// TIA Portal V17 export
// export: Created 2025-05-06T13:48:25.8957092Z, ExportSetting WithDefaults, DisplayName Totally Integrated Automation Portal, DisplayVersion V17 Update 8, DisplayName TIA Portal Openness, DisplayVersion V17 Update 8, DisplayName TIA Portal Version Control Interface, DisplayVersion V17, DisplayName SINAMICS Startdrive Advanced, DisplayVersion V17 SP2, DisplayName SINAMICS Startdrive G110M, G120, G120C, G120D, G120P, G115D, DisplayVersion V17 SP2, DisplayName SINAMICS Startdrive G130, G150, S120, S150, SINAMICS MV, S210, DisplayVersion V17 SP2, DisplayName STEP 7 Professional, DisplayVersion V17 Update 8, DisplayName SINUMERIK ONE STEP 7 Toolbox, DisplayVersion V17 Update 12, DisplayName SINUMERIK 840D sl STEP 7 Toolbox, DisplayVersion V17 Update 12, DisplayName STEP 7 Safety, DisplayVersion V17 Update 6, DisplayName WinCC Advanced, DisplayVersion V17 Update 8
FUNCTION "FC5000_FIX_TABLE_POSITIONS" : Void   // FC5000, LAD
TITLE = FC4000_FIX_TABLE_POSITIONS
{ S7_Optimized_Access := 'TRUE' }
VERSION : 0.1
// stored: AutoNumber false, IsIECCheckEnabled false, SetENOAutomatically false, UDAEnableTagReadback false
   VAR_TEMP
      SENSOR_VALUE_TMP : UInt;
   END_VAR
   VAR_TEMP   // added for the SCL form of the ladder/FBD networks
      _w1 : Bool;
      _w2 : Bool;
      _w3 : Bool;
      _w4 : Bool;
   END_VAR
BEGIN

REGION Network 1: <<<<<<<<<<<<<<<<<<<< UNIT 01 >>>>>>>>>>>>>>>>>>>>
END_REGION

REGION Network 2: AXIS E10 0 DEGREES
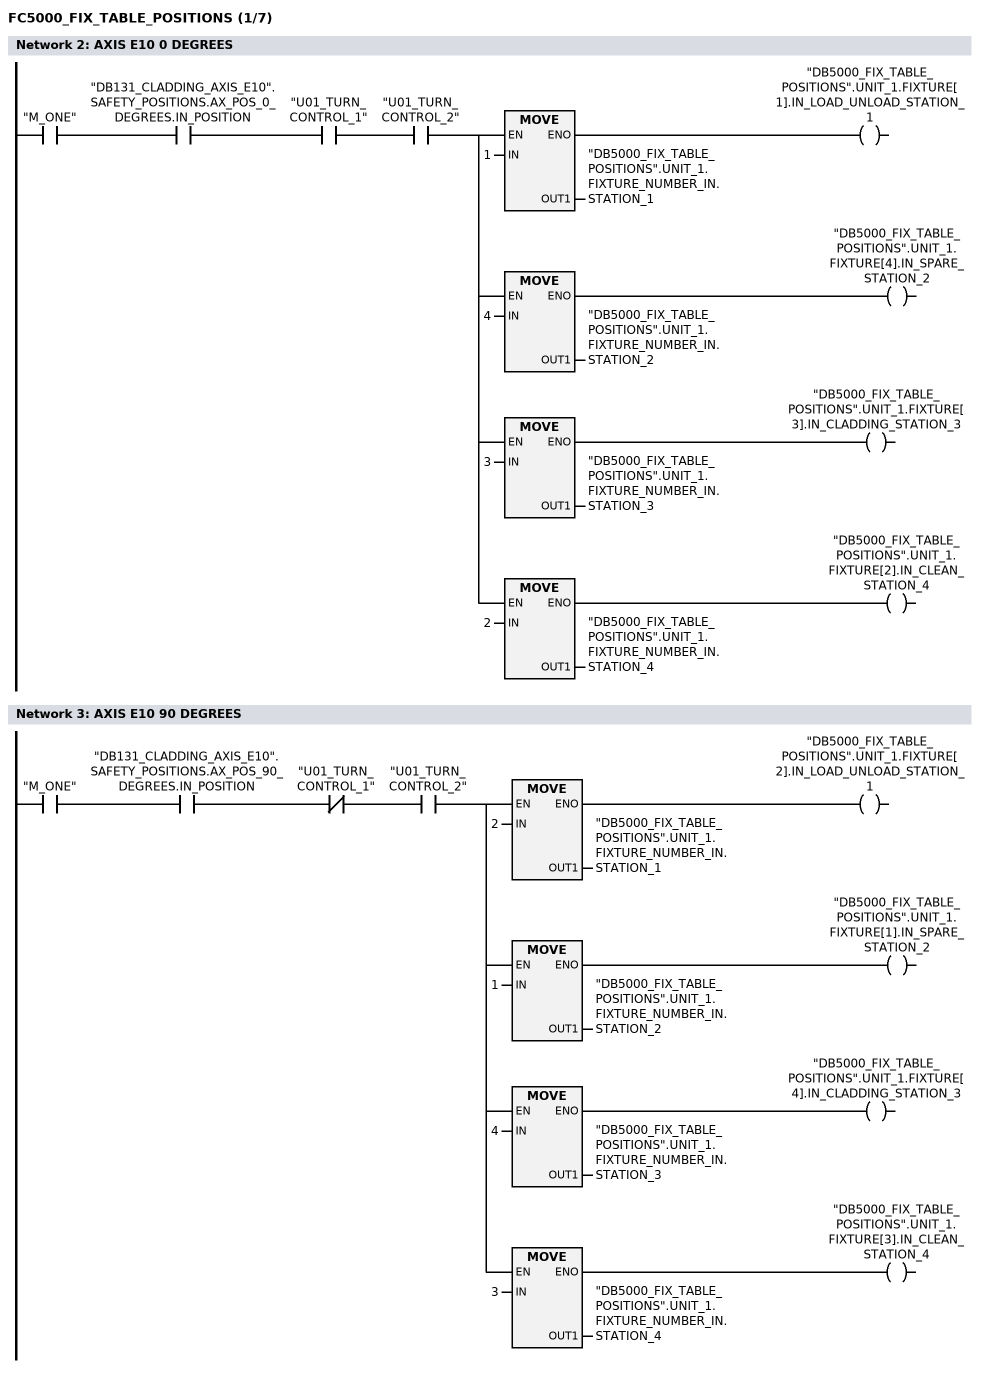
   RUNG wire#powerrail
      Contact( "M_ONE" )
      Contact( "DB131_CLADDING_AXIS_E10".SAFETY_POSITIONS.AX_POS_0_DEGREES.IN_POSITION )
      Contact( "U01_TURN_CONTROL_1" )
      Contact( "U01_TURN_CONTROL_2" )
      wire#w1
      Move(in := 1, out1 => "DB5000_FIX_TABLE_POSITIONS".UNIT_1.FIXTURE_NUMBER_IN.STATION_1)
      Coil( "DB5000_FIX_TABLE_POSITIONS".UNIT_1.FIXTURE[1].IN_LOAD_UNLOAD_STATION_1 )
   END_RUNG
   RUNG wire#w1
      Move(in := 4, out1 => "DB5000_FIX_TABLE_POSITIONS".UNIT_1.FIXTURE_NUMBER_IN.STATION_2)
      Coil( "DB5000_FIX_TABLE_POSITIONS".UNIT_1.FIXTURE[4].IN_SPARE_STATION_2 )
   END_RUNG
   RUNG wire#w1
      Move(in := 3, out1 => "DB5000_FIX_TABLE_POSITIONS".UNIT_1.FIXTURE_NUMBER_IN.STATION_3)
      Coil( "DB5000_FIX_TABLE_POSITIONS".UNIT_1.FIXTURE[3].IN_CLADDING_STATION_3 )
   END_RUNG
   RUNG wire#w1
      Move(in := 2, out1 => "DB5000_FIX_TABLE_POSITIONS".UNIT_1.FIXTURE_NUMBER_IN.STATION_4)
      Coil( "DB5000_FIX_TABLE_POSITIONS".UNIT_1.FIXTURE[2].IN_CLEAN_STATION_4 )
   END_RUNG
   // the same network as SCL:
   #_w1 := "M_ONE" AND "DB131_CLADDING_AXIS_E10".SAFETY_POSITIONS.AX_POS_0_DEGREES.IN_POSITION AND "U01_TURN_CONTROL_1" AND "U01_TURN_CONTROL_2";
   IF #_w1 THEN "DB5000_FIX_TABLE_POSITIONS".UNIT_1.FIXTURE_NUMBER_IN.STATION_1 := 1; END_IF;
   "DB5000_FIX_TABLE_POSITIONS".UNIT_1.FIXTURE[1].IN_LOAD_UNLOAD_STATION_1 := #_w1;
   IF #_w1 THEN "DB5000_FIX_TABLE_POSITIONS".UNIT_1.FIXTURE_NUMBER_IN.STATION_2 := 4; END_IF;
   "DB5000_FIX_TABLE_POSITIONS".UNIT_1.FIXTURE[4].IN_SPARE_STATION_2 := #_w1;
   IF #_w1 THEN "DB5000_FIX_TABLE_POSITIONS".UNIT_1.FIXTURE_NUMBER_IN.STATION_3 := 3; END_IF;
   "DB5000_FIX_TABLE_POSITIONS".UNIT_1.FIXTURE[3].IN_CLADDING_STATION_3 := #_w1;
   IF #_w1 THEN "DB5000_FIX_TABLE_POSITIONS".UNIT_1.FIXTURE_NUMBER_IN.STATION_4 := 2; END_IF;
   "DB5000_FIX_TABLE_POSITIONS".UNIT_1.FIXTURE[2].IN_CLEAN_STATION_4 := #_w1;
END_REGION

REGION Network 3: AXIS E10 90 DEGREES
   RUNG wire#powerrail
      Contact( "M_ONE" )
      Contact( "DB131_CLADDING_AXIS_E10".SAFETY_POSITIONS.AX_POS_90_DEGREES.IN_POSITION )
      I_Contact( "U01_TURN_CONTROL_1" )
      Contact( "U01_TURN_CONTROL_2" )
      wire#w1
      Move(in := 2, out1 => "DB5000_FIX_TABLE_POSITIONS".UNIT_1.FIXTURE_NUMBER_IN.STATION_1)
      Coil( "DB5000_FIX_TABLE_POSITIONS".UNIT_1.FIXTURE[2].IN_LOAD_UNLOAD_STATION_1 )
   END_RUNG
   RUNG wire#w1
      Move(in := 1, out1 => "DB5000_FIX_TABLE_POSITIONS".UNIT_1.FIXTURE_NUMBER_IN.STATION_2)
      Coil( "DB5000_FIX_TABLE_POSITIONS".UNIT_1.FIXTURE[1].IN_SPARE_STATION_2 )
   END_RUNG
   RUNG wire#w1
      Move(in := 4, out1 => "DB5000_FIX_TABLE_POSITIONS".UNIT_1.FIXTURE_NUMBER_IN.STATION_3)
      Coil( "DB5000_FIX_TABLE_POSITIONS".UNIT_1.FIXTURE[4].IN_CLADDING_STATION_3 )
   END_RUNG
   RUNG wire#w1
      Move(in := 3, out1 => "DB5000_FIX_TABLE_POSITIONS".UNIT_1.FIXTURE_NUMBER_IN.STATION_4)
      Coil( "DB5000_FIX_TABLE_POSITIONS".UNIT_1.FIXTURE[3].IN_CLEAN_STATION_4 )
   END_RUNG
   // the same network as SCL:
   #_w1 := "M_ONE" AND "DB131_CLADDING_AXIS_E10".SAFETY_POSITIONS.AX_POS_90_DEGREES.IN_POSITION AND NOT "U01_TURN_CONTROL_1" AND "U01_TURN_CONTROL_2";
   IF #_w1 THEN "DB5000_FIX_TABLE_POSITIONS".UNIT_1.FIXTURE_NUMBER_IN.STATION_1 := 2; END_IF;
   "DB5000_FIX_TABLE_POSITIONS".UNIT_1.FIXTURE[2].IN_LOAD_UNLOAD_STATION_1 := #_w1;
   IF #_w1 THEN "DB5000_FIX_TABLE_POSITIONS".UNIT_1.FIXTURE_NUMBER_IN.STATION_2 := 1; END_IF;
   "DB5000_FIX_TABLE_POSITIONS".UNIT_1.FIXTURE[1].IN_SPARE_STATION_2 := #_w1;
   IF #_w1 THEN "DB5000_FIX_TABLE_POSITIONS".UNIT_1.FIXTURE_NUMBER_IN.STATION_3 := 4; END_IF;
   "DB5000_FIX_TABLE_POSITIONS".UNIT_1.FIXTURE[4].IN_CLADDING_STATION_3 := #_w1;
   IF #_w1 THEN "DB5000_FIX_TABLE_POSITIONS".UNIT_1.FIXTURE_NUMBER_IN.STATION_4 := 3; END_IF;
   "DB5000_FIX_TABLE_POSITIONS".UNIT_1.FIXTURE[3].IN_CLEAN_STATION_4 := #_w1;
END_REGION

REGION Network 4: AXIS E10 180 DEGREES
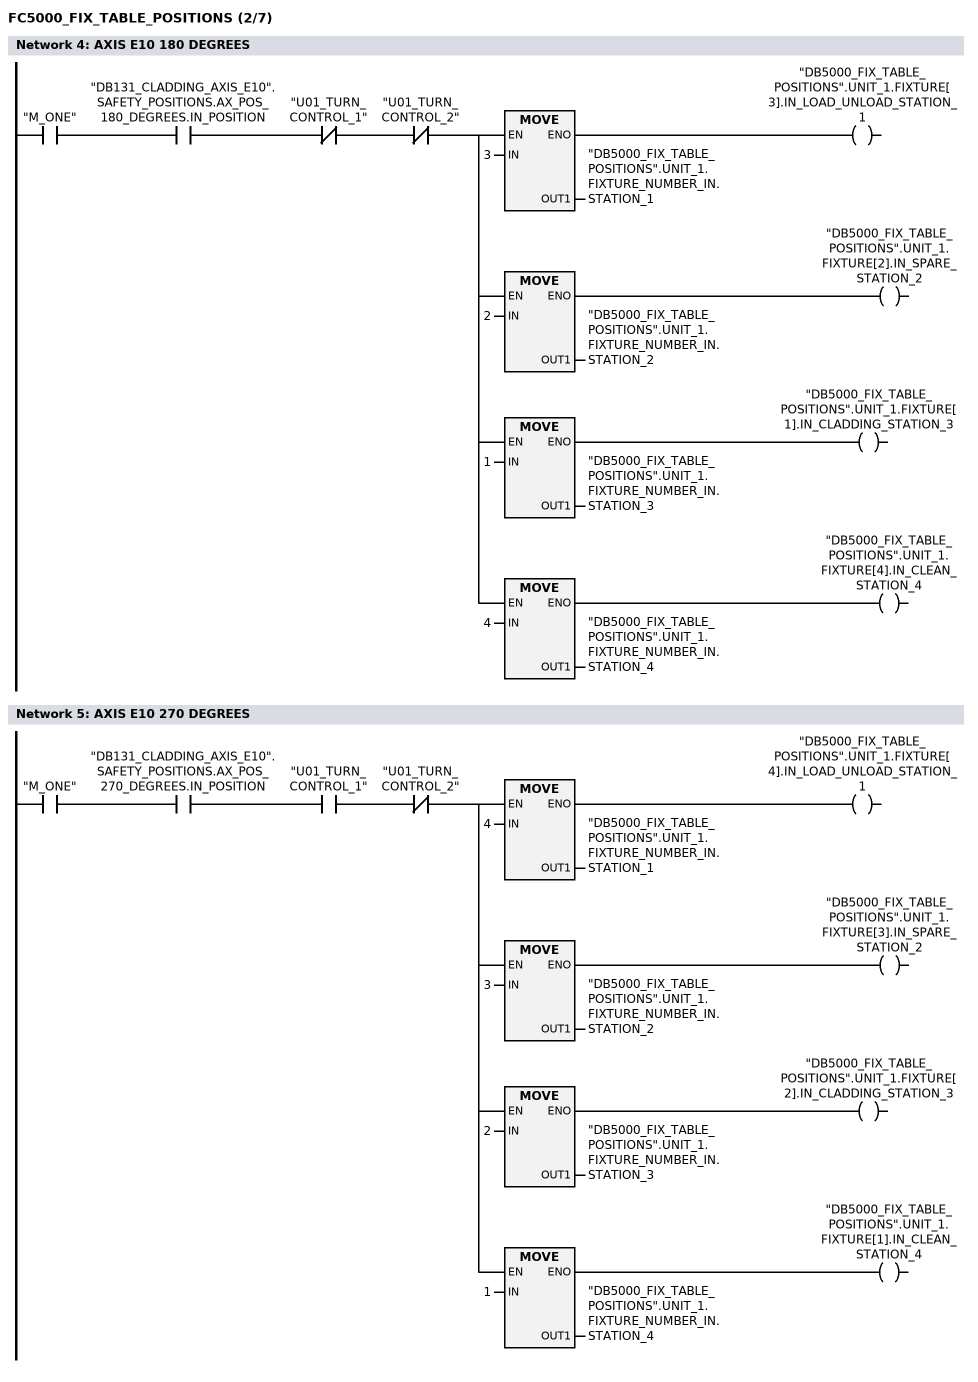
   RUNG wire#powerrail
      Contact( "M_ONE" )
      Contact( "DB131_CLADDING_AXIS_E10".SAFETY_POSITIONS.AX_POS_180_DEGREES.IN_POSITION )
      I_Contact( "U01_TURN_CONTROL_1" )
      I_Contact( "U01_TURN_CONTROL_2" )
      wire#w1
      Move(in := 3, out1 => "DB5000_FIX_TABLE_POSITIONS".UNIT_1.FIXTURE_NUMBER_IN.STATION_1)
      Coil( "DB5000_FIX_TABLE_POSITIONS".UNIT_1.FIXTURE[3].IN_LOAD_UNLOAD_STATION_1 )
   END_RUNG
   RUNG wire#w1
      Move(in := 2, out1 => "DB5000_FIX_TABLE_POSITIONS".UNIT_1.FIXTURE_NUMBER_IN.STATION_2)
      Coil( "DB5000_FIX_TABLE_POSITIONS".UNIT_1.FIXTURE[2].IN_SPARE_STATION_2 )
   END_RUNG
   RUNG wire#w1
      Move(in := 1, out1 => "DB5000_FIX_TABLE_POSITIONS".UNIT_1.FIXTURE_NUMBER_IN.STATION_3)
      Coil( "DB5000_FIX_TABLE_POSITIONS".UNIT_1.FIXTURE[1].IN_CLADDING_STATION_3 )
   END_RUNG
   RUNG wire#w1
      Move(in := 4, out1 => "DB5000_FIX_TABLE_POSITIONS".UNIT_1.FIXTURE_NUMBER_IN.STATION_4)
      Coil( "DB5000_FIX_TABLE_POSITIONS".UNIT_1.FIXTURE[4].IN_CLEAN_STATION_4 )
   END_RUNG
   // the same network as SCL:
   #_w1 := "M_ONE" AND "DB131_CLADDING_AXIS_E10".SAFETY_POSITIONS.AX_POS_180_DEGREES.IN_POSITION AND NOT "U01_TURN_CONTROL_1" AND NOT "U01_TURN_CONTROL_2";
   IF #_w1 THEN "DB5000_FIX_TABLE_POSITIONS".UNIT_1.FIXTURE_NUMBER_IN.STATION_1 := 3; END_IF;
   "DB5000_FIX_TABLE_POSITIONS".UNIT_1.FIXTURE[3].IN_LOAD_UNLOAD_STATION_1 := #_w1;
   IF #_w1 THEN "DB5000_FIX_TABLE_POSITIONS".UNIT_1.FIXTURE_NUMBER_IN.STATION_2 := 2; END_IF;
   "DB5000_FIX_TABLE_POSITIONS".UNIT_1.FIXTURE[2].IN_SPARE_STATION_2 := #_w1;
   IF #_w1 THEN "DB5000_FIX_TABLE_POSITIONS".UNIT_1.FIXTURE_NUMBER_IN.STATION_3 := 1; END_IF;
   "DB5000_FIX_TABLE_POSITIONS".UNIT_1.FIXTURE[1].IN_CLADDING_STATION_3 := #_w1;
   IF #_w1 THEN "DB5000_FIX_TABLE_POSITIONS".UNIT_1.FIXTURE_NUMBER_IN.STATION_4 := 4; END_IF;
   "DB5000_FIX_TABLE_POSITIONS".UNIT_1.FIXTURE[4].IN_CLEAN_STATION_4 := #_w1;
END_REGION

REGION Network 5: AXIS E10 270 DEGREES
   RUNG wire#powerrail
      Contact( "M_ONE" )
      Contact( "DB131_CLADDING_AXIS_E10".SAFETY_POSITIONS.AX_POS_270_DEGREES.IN_POSITION )
      Contact( "U01_TURN_CONTROL_1" )
      I_Contact( "U01_TURN_CONTROL_2" )
      wire#w1
      Move(in := 4, out1 => "DB5000_FIX_TABLE_POSITIONS".UNIT_1.FIXTURE_NUMBER_IN.STATION_1)
      Coil( "DB5000_FIX_TABLE_POSITIONS".UNIT_1.FIXTURE[4].IN_LOAD_UNLOAD_STATION_1 )
   END_RUNG
   RUNG wire#w1
      Move(in := 3, out1 => "DB5000_FIX_TABLE_POSITIONS".UNIT_1.FIXTURE_NUMBER_IN.STATION_2)
      Coil( "DB5000_FIX_TABLE_POSITIONS".UNIT_1.FIXTURE[3].IN_SPARE_STATION_2 )
   END_RUNG
   RUNG wire#w1
      Move(in := 2, out1 => "DB5000_FIX_TABLE_POSITIONS".UNIT_1.FIXTURE_NUMBER_IN.STATION_3)
      Coil( "DB5000_FIX_TABLE_POSITIONS".UNIT_1.FIXTURE[2].IN_CLADDING_STATION_3 )
   END_RUNG
   RUNG wire#w1
      Move(in := 1, out1 => "DB5000_FIX_TABLE_POSITIONS".UNIT_1.FIXTURE_NUMBER_IN.STATION_4)
      Coil( "DB5000_FIX_TABLE_POSITIONS".UNIT_1.FIXTURE[1].IN_CLEAN_STATION_4 )
   END_RUNG
   // the same network as SCL:
   #_w1 := "M_ONE" AND "DB131_CLADDING_AXIS_E10".SAFETY_POSITIONS.AX_POS_270_DEGREES.IN_POSITION AND "U01_TURN_CONTROL_1" AND NOT "U01_TURN_CONTROL_2";
   IF #_w1 THEN "DB5000_FIX_TABLE_POSITIONS".UNIT_1.FIXTURE_NUMBER_IN.STATION_1 := 4; END_IF;
   "DB5000_FIX_TABLE_POSITIONS".UNIT_1.FIXTURE[4].IN_LOAD_UNLOAD_STATION_1 := #_w1;
   IF #_w1 THEN "DB5000_FIX_TABLE_POSITIONS".UNIT_1.FIXTURE_NUMBER_IN.STATION_2 := 3; END_IF;
   "DB5000_FIX_TABLE_POSITIONS".UNIT_1.FIXTURE[3].IN_SPARE_STATION_2 := #_w1;
   IF #_w1 THEN "DB5000_FIX_TABLE_POSITIONS".UNIT_1.FIXTURE_NUMBER_IN.STATION_3 := 2; END_IF;
   "DB5000_FIX_TABLE_POSITIONS".UNIT_1.FIXTURE[2].IN_CLADDING_STATION_3 := #_w1;
   IF #_w1 THEN "DB5000_FIX_TABLE_POSITIONS".UNIT_1.FIXTURE_NUMBER_IN.STATION_4 := 1; END_IF;
   "DB5000_FIX_TABLE_POSITIONS".UNIT_1.FIXTURE[1].IN_CLEAN_STATION_4 := #_w1;
END_REGION

REGION Network 6: E10 AXIS POSITION REACH
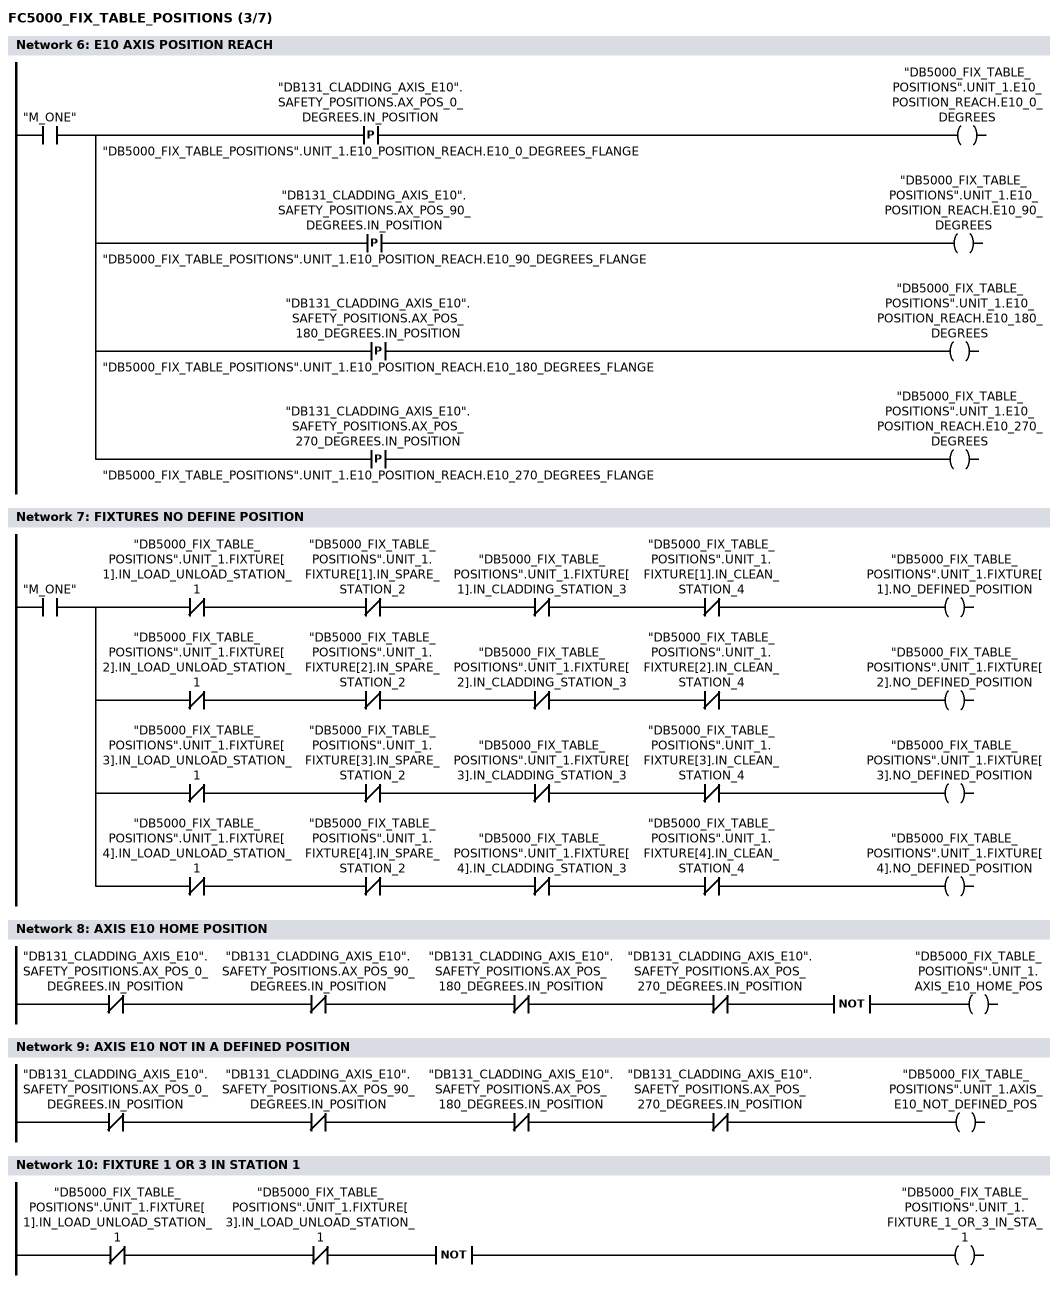
   RUNG wire#powerrail
      Contact( "M_ONE" )
      wire#w1
      P_Contact(operand := "DB131_CLADDING_AXIS_E10".SAFETY_POSITIONS.AX_POS_0_DEGREES.IN_POSITION, bit := "DB5000_FIX_TABLE_POSITIONS".UNIT_1.E10_POSITION_REACH.E10_0_DEGREES_FLANGE)
      Coil( "DB5000_FIX_TABLE_POSITIONS".UNIT_1.E10_POSITION_REACH.E10_0_DEGREES )
   END_RUNG
   RUNG wire#w1
      P_Contact(operand := "DB131_CLADDING_AXIS_E10".SAFETY_POSITIONS.AX_POS_90_DEGREES.IN_POSITION, bit := "DB5000_FIX_TABLE_POSITIONS".UNIT_1.E10_POSITION_REACH.E10_90_DEGREES_FLANGE)
      Coil( "DB5000_FIX_TABLE_POSITIONS".UNIT_1.E10_POSITION_REACH.E10_90_DEGREES )
   END_RUNG
   RUNG wire#w1
      P_Contact(operand := "DB131_CLADDING_AXIS_E10".SAFETY_POSITIONS.AX_POS_180_DEGREES.IN_POSITION, bit := "DB5000_FIX_TABLE_POSITIONS".UNIT_1.E10_POSITION_REACH.E10_180_DEGREES_FLANGE)
      Coil( "DB5000_FIX_TABLE_POSITIONS".UNIT_1.E10_POSITION_REACH.E10_180_DEGREES )
   END_RUNG
   RUNG wire#w1
      P_Contact(operand := "DB131_CLADDING_AXIS_E10".SAFETY_POSITIONS.AX_POS_270_DEGREES.IN_POSITION, bit := "DB5000_FIX_TABLE_POSITIONS".UNIT_1.E10_POSITION_REACH.E10_270_DEGREES_FLANGE)
      Coil( "DB5000_FIX_TABLE_POSITIONS".UNIT_1.E10_POSITION_REACH.E10_270_DEGREES )
   END_RUNG
   // the same network as SCL:
   #_w1 := "M_ONE" AND "DB131_CLADDING_AXIS_E10".SAFETY_POSITIONS.AX_POS_0_DEGREES.IN_POSITION AND NOT "DB5000_FIX_TABLE_POSITIONS".UNIT_1.E10_POSITION_REACH.E10_0_DEGREES_FLANGE;   // rising edge of "DB131_CLADDING_AXIS_E10".SAFETY_POSITIONS.AX_POS_0_DEGREES.IN_POSITION
   "DB5000_FIX_TABLE_POSITIONS".UNIT_1.E10_POSITION_REACH.E10_0_DEGREES_FLANGE := "DB131_CLADDING_AXIS_E10".SAFETY_POSITIONS.AX_POS_0_DEGREES.IN_POSITION;
   "DB5000_FIX_TABLE_POSITIONS".UNIT_1.E10_POSITION_REACH.E10_0_DEGREES := #_w1;
   #_w2 := "M_ONE" AND "DB131_CLADDING_AXIS_E10".SAFETY_POSITIONS.AX_POS_90_DEGREES.IN_POSITION AND NOT "DB5000_FIX_TABLE_POSITIONS".UNIT_1.E10_POSITION_REACH.E10_90_DEGREES_FLANGE;   // rising edge of "DB131_CLADDING_AXIS_E10".SAFETY_POSITIONS.AX_POS_90_DEGREES.IN_POSITION
   "DB5000_FIX_TABLE_POSITIONS".UNIT_1.E10_POSITION_REACH.E10_90_DEGREES_FLANGE := "DB131_CLADDING_AXIS_E10".SAFETY_POSITIONS.AX_POS_90_DEGREES.IN_POSITION;
   "DB5000_FIX_TABLE_POSITIONS".UNIT_1.E10_POSITION_REACH.E10_90_DEGREES := #_w2;
   #_w3 := "M_ONE" AND "DB131_CLADDING_AXIS_E10".SAFETY_POSITIONS.AX_POS_180_DEGREES.IN_POSITION AND NOT "DB5000_FIX_TABLE_POSITIONS".UNIT_1.E10_POSITION_REACH.E10_180_DEGREES_FLANGE;   // rising edge of "DB131_CLADDING_AXIS_E10".SAFETY_POSITIONS.AX_POS_180_DEGREES.IN_POSITION
   "DB5000_FIX_TABLE_POSITIONS".UNIT_1.E10_POSITION_REACH.E10_180_DEGREES_FLANGE := "DB131_CLADDING_AXIS_E10".SAFETY_POSITIONS.AX_POS_180_DEGREES.IN_POSITION;
   "DB5000_FIX_TABLE_POSITIONS".UNIT_1.E10_POSITION_REACH.E10_180_DEGREES := #_w3;
   #_w4 := "M_ONE" AND "DB131_CLADDING_AXIS_E10".SAFETY_POSITIONS.AX_POS_270_DEGREES.IN_POSITION AND NOT "DB5000_FIX_TABLE_POSITIONS".UNIT_1.E10_POSITION_REACH.E10_270_DEGREES_FLANGE;   // rising edge of "DB131_CLADDING_AXIS_E10".SAFETY_POSITIONS.AX_POS_270_DEGREES.IN_POSITION
   "DB5000_FIX_TABLE_POSITIONS".UNIT_1.E10_POSITION_REACH.E10_270_DEGREES_FLANGE := "DB131_CLADDING_AXIS_E10".SAFETY_POSITIONS.AX_POS_270_DEGREES.IN_POSITION;
   "DB5000_FIX_TABLE_POSITIONS".UNIT_1.E10_POSITION_REACH.E10_270_DEGREES := #_w4;
END_REGION

REGION Network 7: FIXTURES NO DEFINE POSITION
   RUNG wire#powerrail
      Contact( "M_ONE" )
      wire#w1
      I_Contact( "DB5000_FIX_TABLE_POSITIONS".UNIT_1.FIXTURE[1].IN_LOAD_UNLOAD_STATION_1 )
      I_Contact( "DB5000_FIX_TABLE_POSITIONS".UNIT_1.FIXTURE[1].IN_SPARE_STATION_2 )
      I_Contact( "DB5000_FIX_TABLE_POSITIONS".UNIT_1.FIXTURE[1].IN_CLADDING_STATION_3 )
      I_Contact( "DB5000_FIX_TABLE_POSITIONS".UNIT_1.FIXTURE[1].IN_CLEAN_STATION_4 )
      Coil( "DB5000_FIX_TABLE_POSITIONS".UNIT_1.FIXTURE[1].NO_DEFINED_POSITION )
   END_RUNG
   RUNG wire#w1
      I_Contact( "DB5000_FIX_TABLE_POSITIONS".UNIT_1.FIXTURE[2].IN_LOAD_UNLOAD_STATION_1 )
      I_Contact( "DB5000_FIX_TABLE_POSITIONS".UNIT_1.FIXTURE[2].IN_SPARE_STATION_2 )
      I_Contact( "DB5000_FIX_TABLE_POSITIONS".UNIT_1.FIXTURE[2].IN_CLADDING_STATION_3 )
      I_Contact( "DB5000_FIX_TABLE_POSITIONS".UNIT_1.FIXTURE[2].IN_CLEAN_STATION_4 )
      Coil( "DB5000_FIX_TABLE_POSITIONS".UNIT_1.FIXTURE[2].NO_DEFINED_POSITION )
   END_RUNG
   RUNG wire#w1
      I_Contact( "DB5000_FIX_TABLE_POSITIONS".UNIT_1.FIXTURE[3].IN_LOAD_UNLOAD_STATION_1 )
      I_Contact( "DB5000_FIX_TABLE_POSITIONS".UNIT_1.FIXTURE[3].IN_SPARE_STATION_2 )
      I_Contact( "DB5000_FIX_TABLE_POSITIONS".UNIT_1.FIXTURE[3].IN_CLADDING_STATION_3 )
      I_Contact( "DB5000_FIX_TABLE_POSITIONS".UNIT_1.FIXTURE[3].IN_CLEAN_STATION_4 )
      Coil( "DB5000_FIX_TABLE_POSITIONS".UNIT_1.FIXTURE[3].NO_DEFINED_POSITION )
   END_RUNG
   RUNG wire#w1
      I_Contact( "DB5000_FIX_TABLE_POSITIONS".UNIT_1.FIXTURE[4].IN_LOAD_UNLOAD_STATION_1 )
      I_Contact( "DB5000_FIX_TABLE_POSITIONS".UNIT_1.FIXTURE[4].IN_SPARE_STATION_2 )
      I_Contact( "DB5000_FIX_TABLE_POSITIONS".UNIT_1.FIXTURE[4].IN_CLADDING_STATION_3 )
      I_Contact( "DB5000_FIX_TABLE_POSITIONS".UNIT_1.FIXTURE[4].IN_CLEAN_STATION_4 )
      Coil( "DB5000_FIX_TABLE_POSITIONS".UNIT_1.FIXTURE[4].NO_DEFINED_POSITION )
   END_RUNG
   // the same network as SCL:
   "DB5000_FIX_TABLE_POSITIONS".UNIT_1.FIXTURE[1].NO_DEFINED_POSITION := "M_ONE" AND NOT "DB5000_FIX_TABLE_POSITIONS".UNIT_1.FIXTURE[1].IN_LOAD_UNLOAD_STATION_1 AND NOT "DB5000_FIX_TABLE_POSITIONS".UNIT_1.FIXTURE[1].IN_SPARE_STATION_2 AND NOT "DB5000_FIX_TABLE_POSITIONS".UNIT_1.FIXTURE[1].IN_CLADDING_STATION_3 AND NOT "DB5000_FIX_TABLE_POSITIONS".UNIT_1.FIXTURE[1].IN_CLEAN_STATION_4;
   "DB5000_FIX_TABLE_POSITIONS".UNIT_1.FIXTURE[2].NO_DEFINED_POSITION := "M_ONE" AND NOT "DB5000_FIX_TABLE_POSITIONS".UNIT_1.FIXTURE[2].IN_LOAD_UNLOAD_STATION_1 AND NOT "DB5000_FIX_TABLE_POSITIONS".UNIT_1.FIXTURE[2].IN_SPARE_STATION_2 AND NOT "DB5000_FIX_TABLE_POSITIONS".UNIT_1.FIXTURE[2].IN_CLADDING_STATION_3 AND NOT "DB5000_FIX_TABLE_POSITIONS".UNIT_1.FIXTURE[2].IN_CLEAN_STATION_4;
   "DB5000_FIX_TABLE_POSITIONS".UNIT_1.FIXTURE[3].NO_DEFINED_POSITION := "M_ONE" AND NOT "DB5000_FIX_TABLE_POSITIONS".UNIT_1.FIXTURE[3].IN_LOAD_UNLOAD_STATION_1 AND NOT "DB5000_FIX_TABLE_POSITIONS".UNIT_1.FIXTURE[3].IN_SPARE_STATION_2 AND NOT "DB5000_FIX_TABLE_POSITIONS".UNIT_1.FIXTURE[3].IN_CLADDING_STATION_3 AND NOT "DB5000_FIX_TABLE_POSITIONS".UNIT_1.FIXTURE[3].IN_CLEAN_STATION_4;
   "DB5000_FIX_TABLE_POSITIONS".UNIT_1.FIXTURE[4].NO_DEFINED_POSITION := "M_ONE" AND NOT "DB5000_FIX_TABLE_POSITIONS".UNIT_1.FIXTURE[4].IN_LOAD_UNLOAD_STATION_1 AND NOT "DB5000_FIX_TABLE_POSITIONS".UNIT_1.FIXTURE[4].IN_SPARE_STATION_2 AND NOT "DB5000_FIX_TABLE_POSITIONS".UNIT_1.FIXTURE[4].IN_CLADDING_STATION_3 AND NOT "DB5000_FIX_TABLE_POSITIONS".UNIT_1.FIXTURE[4].IN_CLEAN_STATION_4;
END_REGION

REGION Network 8: AXIS E10 HOME POSITION
   RUNG wire#powerrail
      I_Contact( "DB131_CLADDING_AXIS_E10".SAFETY_POSITIONS.AX_POS_0_DEGREES.IN_POSITION )
      I_Contact( "DB131_CLADDING_AXIS_E10".SAFETY_POSITIONS.AX_POS_90_DEGREES.IN_POSITION )
      I_Contact( "DB131_CLADDING_AXIS_E10".SAFETY_POSITIONS.AX_POS_180_DEGREES.IN_POSITION )
      I_Contact( "DB131_CLADDING_AXIS_E10".SAFETY_POSITIONS.AX_POS_270_DEGREES.IN_POSITION )
      Not()
      Coil( "DB5000_FIX_TABLE_POSITIONS".UNIT_1.AXIS_E10_HOME_POS )
   END_RUNG
   // the same network as SCL:
   "DB5000_FIX_TABLE_POSITIONS".UNIT_1.AXIS_E10_HOME_POS := NOT (NOT "DB131_CLADDING_AXIS_E10".SAFETY_POSITIONS.AX_POS_0_DEGREES.IN_POSITION AND NOT "DB131_CLADDING_AXIS_E10".SAFETY_POSITIONS.AX_POS_90_DEGREES.IN_POSITION AND NOT "DB131_CLADDING_AXIS_E10".SAFETY_POSITIONS.AX_POS_180_DEGREES.IN_POSITION AND NOT "DB131_CLADDING_AXIS_E10".SAFETY_POSITIONS.AX_POS_270_DEGREES.IN_POSITION);
END_REGION

REGION Network 9: AXIS E10 NOT IN A DEFINED POSITION
   RUNG wire#powerrail
      I_Contact( "DB131_CLADDING_AXIS_E10".SAFETY_POSITIONS.AX_POS_0_DEGREES.IN_POSITION )
      I_Contact( "DB131_CLADDING_AXIS_E10".SAFETY_POSITIONS.AX_POS_90_DEGREES.IN_POSITION )
      I_Contact( "DB131_CLADDING_AXIS_E10".SAFETY_POSITIONS.AX_POS_180_DEGREES.IN_POSITION )
      I_Contact( "DB131_CLADDING_AXIS_E10".SAFETY_POSITIONS.AX_POS_270_DEGREES.IN_POSITION )
      Coil( "DB5000_FIX_TABLE_POSITIONS".UNIT_1.AXIS_E10_NOT_DEFINED_POS )
   END_RUNG
   // the same network as SCL:
   "DB5000_FIX_TABLE_POSITIONS".UNIT_1.AXIS_E10_NOT_DEFINED_POS := NOT "DB131_CLADDING_AXIS_E10".SAFETY_POSITIONS.AX_POS_0_DEGREES.IN_POSITION AND NOT "DB131_CLADDING_AXIS_E10".SAFETY_POSITIONS.AX_POS_90_DEGREES.IN_POSITION AND NOT "DB131_CLADDING_AXIS_E10".SAFETY_POSITIONS.AX_POS_180_DEGREES.IN_POSITION AND NOT "DB131_CLADDING_AXIS_E10".SAFETY_POSITIONS.AX_POS_270_DEGREES.IN_POSITION;
END_REGION

REGION Network 10: FIXTURE 1 OR 3 IN STATION 1
   RUNG wire#powerrail
      I_Contact( "DB5000_FIX_TABLE_POSITIONS".UNIT_1.FIXTURE[1].IN_LOAD_UNLOAD_STATION_1 )
      I_Contact( "DB5000_FIX_TABLE_POSITIONS".UNIT_1.FIXTURE[3].IN_LOAD_UNLOAD_STATION_1 )
      Not()
      Coil( "DB5000_FIX_TABLE_POSITIONS".UNIT_1.FIXTURE_1_OR_3_IN_STA_1 )
   END_RUNG
   // the same network as SCL:
   "DB5000_FIX_TABLE_POSITIONS".UNIT_1.FIXTURE_1_OR_3_IN_STA_1 := NOT (NOT "DB5000_FIX_TABLE_POSITIONS".UNIT_1.FIXTURE[1].IN_LOAD_UNLOAD_STATION_1 AND NOT "DB5000_FIX_TABLE_POSITIONS".UNIT_1.FIXTURE[3].IN_LOAD_UNLOAD_STATION_1);
END_REGION

REGION Network 11: FIXTURE 2 OR 4 IN STATION 1
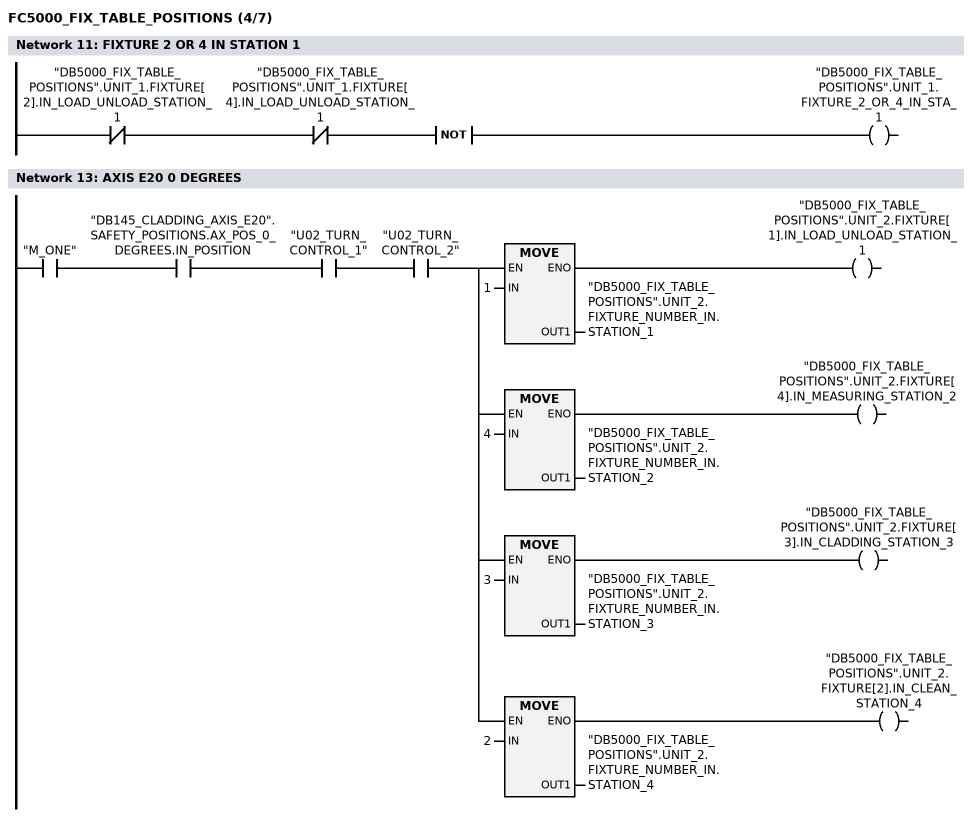
   RUNG wire#powerrail
      I_Contact( "DB5000_FIX_TABLE_POSITIONS".UNIT_1.FIXTURE[2].IN_LOAD_UNLOAD_STATION_1 )
      I_Contact( "DB5000_FIX_TABLE_POSITIONS".UNIT_1.FIXTURE[4].IN_LOAD_UNLOAD_STATION_1 )
      Not()
      Coil( "DB5000_FIX_TABLE_POSITIONS".UNIT_1.FIXTURE_2_OR_4_IN_STA_1 )
   END_RUNG
   // the same network as SCL:
   "DB5000_FIX_TABLE_POSITIONS".UNIT_1.FIXTURE_2_OR_4_IN_STA_1 := NOT (NOT "DB5000_FIX_TABLE_POSITIONS".UNIT_1.FIXTURE[2].IN_LOAD_UNLOAD_STATION_1 AND NOT "DB5000_FIX_TABLE_POSITIONS".UNIT_1.FIXTURE[4].IN_LOAD_UNLOAD_STATION_1);
END_REGION

REGION Network 12: <<<<<<<<<<<<<<<<<<<< UNIT 02 >>>>>>>>>>>>>>>>>>>>
END_REGION

REGION Network 13: AXIS E20 0 DEGREES
   RUNG wire#powerrail
      Contact( "M_ONE" )
      Contact( "DB145_CLADDING_AXIS_E20".SAFETY_POSITIONS.AX_POS_0_DEGREES.IN_POSITION )
      Contact( "U02_TURN_CONTROL_1" )
      Contact( "U02_TURN_CONTROL_2" )
      wire#w1
      Move(in := 1, out1 => "DB5000_FIX_TABLE_POSITIONS".UNIT_2.FIXTURE_NUMBER_IN.STATION_1)
      Coil( "DB5000_FIX_TABLE_POSITIONS".UNIT_2.FIXTURE[1].IN_LOAD_UNLOAD_STATION_1 )
   END_RUNG
   RUNG wire#w1
      Move(in := 4, out1 => "DB5000_FIX_TABLE_POSITIONS".UNIT_2.FIXTURE_NUMBER_IN.STATION_2)
      Coil( "DB5000_FIX_TABLE_POSITIONS".UNIT_2.FIXTURE[4].IN_MEASURING_STATION_2 )
   END_RUNG
   RUNG wire#w1
      Move(in := 3, out1 => "DB5000_FIX_TABLE_POSITIONS".UNIT_2.FIXTURE_NUMBER_IN.STATION_3)
      Coil( "DB5000_FIX_TABLE_POSITIONS".UNIT_2.FIXTURE[3].IN_CLADDING_STATION_3 )
   END_RUNG
   RUNG wire#w1
      Move(in := 2, out1 => "DB5000_FIX_TABLE_POSITIONS".UNIT_2.FIXTURE_NUMBER_IN.STATION_4)
      Coil( "DB5000_FIX_TABLE_POSITIONS".UNIT_2.FIXTURE[2].IN_CLEAN_STATION_4 )
   END_RUNG
   // the same network as SCL:
   #_w1 := "M_ONE" AND "DB145_CLADDING_AXIS_E20".SAFETY_POSITIONS.AX_POS_0_DEGREES.IN_POSITION AND "U02_TURN_CONTROL_1" AND "U02_TURN_CONTROL_2";
   IF #_w1 THEN "DB5000_FIX_TABLE_POSITIONS".UNIT_2.FIXTURE_NUMBER_IN.STATION_1 := 1; END_IF;
   "DB5000_FIX_TABLE_POSITIONS".UNIT_2.FIXTURE[1].IN_LOAD_UNLOAD_STATION_1 := #_w1;
   IF #_w1 THEN "DB5000_FIX_TABLE_POSITIONS".UNIT_2.FIXTURE_NUMBER_IN.STATION_2 := 4; END_IF;
   "DB5000_FIX_TABLE_POSITIONS".UNIT_2.FIXTURE[4].IN_MEASURING_STATION_2 := #_w1;
   IF #_w1 THEN "DB5000_FIX_TABLE_POSITIONS".UNIT_2.FIXTURE_NUMBER_IN.STATION_3 := 3; END_IF;
   "DB5000_FIX_TABLE_POSITIONS".UNIT_2.FIXTURE[3].IN_CLADDING_STATION_3 := #_w1;
   IF #_w1 THEN "DB5000_FIX_TABLE_POSITIONS".UNIT_2.FIXTURE_NUMBER_IN.STATION_4 := 2; END_IF;
   "DB5000_FIX_TABLE_POSITIONS".UNIT_2.FIXTURE[2].IN_CLEAN_STATION_4 := #_w1;
END_REGION

REGION Network 14: AXIS E20 90 DEGREES
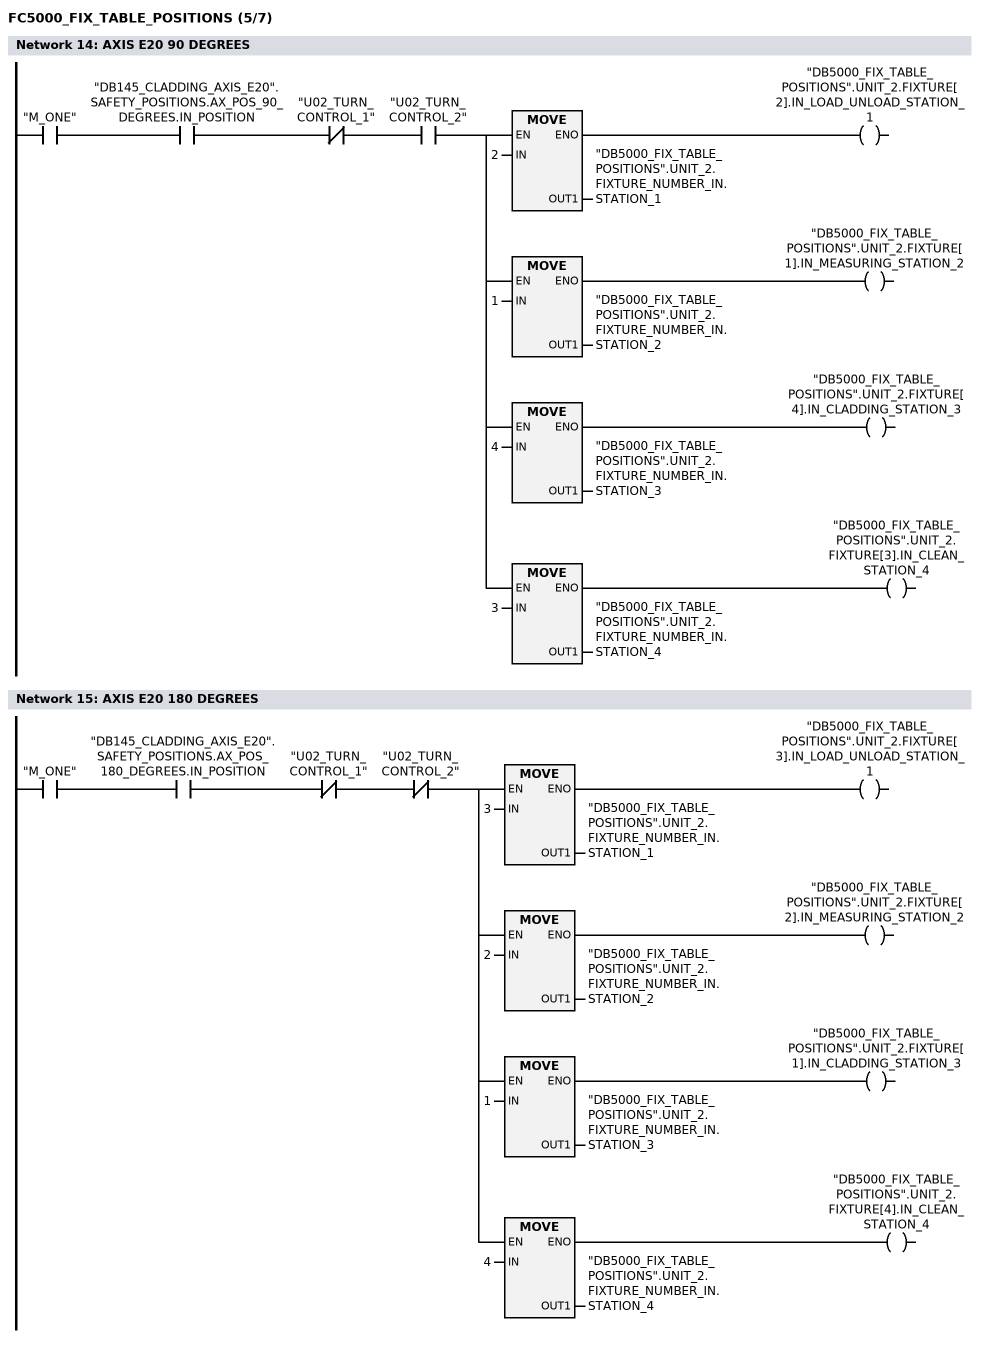
   RUNG wire#powerrail
      Contact( "M_ONE" )
      Contact( "DB145_CLADDING_AXIS_E20".SAFETY_POSITIONS.AX_POS_90_DEGREES.IN_POSITION )
      I_Contact( "U02_TURN_CONTROL_1" )
      Contact( "U02_TURN_CONTROL_2" )
      wire#w1
      Move(in := 2, out1 => "DB5000_FIX_TABLE_POSITIONS".UNIT_2.FIXTURE_NUMBER_IN.STATION_1)
      Coil( "DB5000_FIX_TABLE_POSITIONS".UNIT_2.FIXTURE[2].IN_LOAD_UNLOAD_STATION_1 )
   END_RUNG
   RUNG wire#w1
      Move(in := 1, out1 => "DB5000_FIX_TABLE_POSITIONS".UNIT_2.FIXTURE_NUMBER_IN.STATION_2)
      Coil( "DB5000_FIX_TABLE_POSITIONS".UNIT_2.FIXTURE[1].IN_MEASURING_STATION_2 )
   END_RUNG
   RUNG wire#w1
      Move(in := 4, out1 => "DB5000_FIX_TABLE_POSITIONS".UNIT_2.FIXTURE_NUMBER_IN.STATION_3)
      Coil( "DB5000_FIX_TABLE_POSITIONS".UNIT_2.FIXTURE[4].IN_CLADDING_STATION_3 )
   END_RUNG
   RUNG wire#w1
      Move(in := 3, out1 => "DB5000_FIX_TABLE_POSITIONS".UNIT_2.FIXTURE_NUMBER_IN.STATION_4)
      Coil( "DB5000_FIX_TABLE_POSITIONS".UNIT_2.FIXTURE[3].IN_CLEAN_STATION_4 )
   END_RUNG
   // the same network as SCL:
   #_w1 := "M_ONE" AND "DB145_CLADDING_AXIS_E20".SAFETY_POSITIONS.AX_POS_90_DEGREES.IN_POSITION AND NOT "U02_TURN_CONTROL_1" AND "U02_TURN_CONTROL_2";
   IF #_w1 THEN "DB5000_FIX_TABLE_POSITIONS".UNIT_2.FIXTURE_NUMBER_IN.STATION_1 := 2; END_IF;
   "DB5000_FIX_TABLE_POSITIONS".UNIT_2.FIXTURE[2].IN_LOAD_UNLOAD_STATION_1 := #_w1;
   IF #_w1 THEN "DB5000_FIX_TABLE_POSITIONS".UNIT_2.FIXTURE_NUMBER_IN.STATION_2 := 1; END_IF;
   "DB5000_FIX_TABLE_POSITIONS".UNIT_2.FIXTURE[1].IN_MEASURING_STATION_2 := #_w1;
   IF #_w1 THEN "DB5000_FIX_TABLE_POSITIONS".UNIT_2.FIXTURE_NUMBER_IN.STATION_3 := 4; END_IF;
   "DB5000_FIX_TABLE_POSITIONS".UNIT_2.FIXTURE[4].IN_CLADDING_STATION_3 := #_w1;
   IF #_w1 THEN "DB5000_FIX_TABLE_POSITIONS".UNIT_2.FIXTURE_NUMBER_IN.STATION_4 := 3; END_IF;
   "DB5000_FIX_TABLE_POSITIONS".UNIT_2.FIXTURE[3].IN_CLEAN_STATION_4 := #_w1;
END_REGION

REGION Network 15: AXIS E20 180 DEGREES
   RUNG wire#powerrail
      Contact( "M_ONE" )
      Contact( "DB145_CLADDING_AXIS_E20".SAFETY_POSITIONS.AX_POS_180_DEGREES.IN_POSITION )
      I_Contact( "U02_TURN_CONTROL_1" )
      I_Contact( "U02_TURN_CONTROL_2" )
      wire#w1
      Move(in := 3, out1 => "DB5000_FIX_TABLE_POSITIONS".UNIT_2.FIXTURE_NUMBER_IN.STATION_1)
      Coil( "DB5000_FIX_TABLE_POSITIONS".UNIT_2.FIXTURE[3].IN_LOAD_UNLOAD_STATION_1 )
   END_RUNG
   RUNG wire#w1
      Move(in := 2, out1 => "DB5000_FIX_TABLE_POSITIONS".UNIT_2.FIXTURE_NUMBER_IN.STATION_2)
      Coil( "DB5000_FIX_TABLE_POSITIONS".UNIT_2.FIXTURE[2].IN_MEASURING_STATION_2 )
   END_RUNG
   RUNG wire#w1
      Move(in := 1, out1 => "DB5000_FIX_TABLE_POSITIONS".UNIT_2.FIXTURE_NUMBER_IN.STATION_3)
      Coil( "DB5000_FIX_TABLE_POSITIONS".UNIT_2.FIXTURE[1].IN_CLADDING_STATION_3 )
   END_RUNG
   RUNG wire#w1
      Move(in := 4, out1 => "DB5000_FIX_TABLE_POSITIONS".UNIT_2.FIXTURE_NUMBER_IN.STATION_4)
      Coil( "DB5000_FIX_TABLE_POSITIONS".UNIT_2.FIXTURE[4].IN_CLEAN_STATION_4 )
   END_RUNG
   // the same network as SCL:
   #_w1 := "M_ONE" AND "DB145_CLADDING_AXIS_E20".SAFETY_POSITIONS.AX_POS_180_DEGREES.IN_POSITION AND NOT "U02_TURN_CONTROL_1" AND NOT "U02_TURN_CONTROL_2";
   IF #_w1 THEN "DB5000_FIX_TABLE_POSITIONS".UNIT_2.FIXTURE_NUMBER_IN.STATION_1 := 3; END_IF;
   "DB5000_FIX_TABLE_POSITIONS".UNIT_2.FIXTURE[3].IN_LOAD_UNLOAD_STATION_1 := #_w1;
   IF #_w1 THEN "DB5000_FIX_TABLE_POSITIONS".UNIT_2.FIXTURE_NUMBER_IN.STATION_2 := 2; END_IF;
   "DB5000_FIX_TABLE_POSITIONS".UNIT_2.FIXTURE[2].IN_MEASURING_STATION_2 := #_w1;
   IF #_w1 THEN "DB5000_FIX_TABLE_POSITIONS".UNIT_2.FIXTURE_NUMBER_IN.STATION_3 := 1; END_IF;
   "DB5000_FIX_TABLE_POSITIONS".UNIT_2.FIXTURE[1].IN_CLADDING_STATION_3 := #_w1;
   IF #_w1 THEN "DB5000_FIX_TABLE_POSITIONS".UNIT_2.FIXTURE_NUMBER_IN.STATION_4 := 4; END_IF;
   "DB5000_FIX_TABLE_POSITIONS".UNIT_2.FIXTURE[4].IN_CLEAN_STATION_4 := #_w1;
END_REGION

REGION Network 16: AXIS E20 270 DEGREES
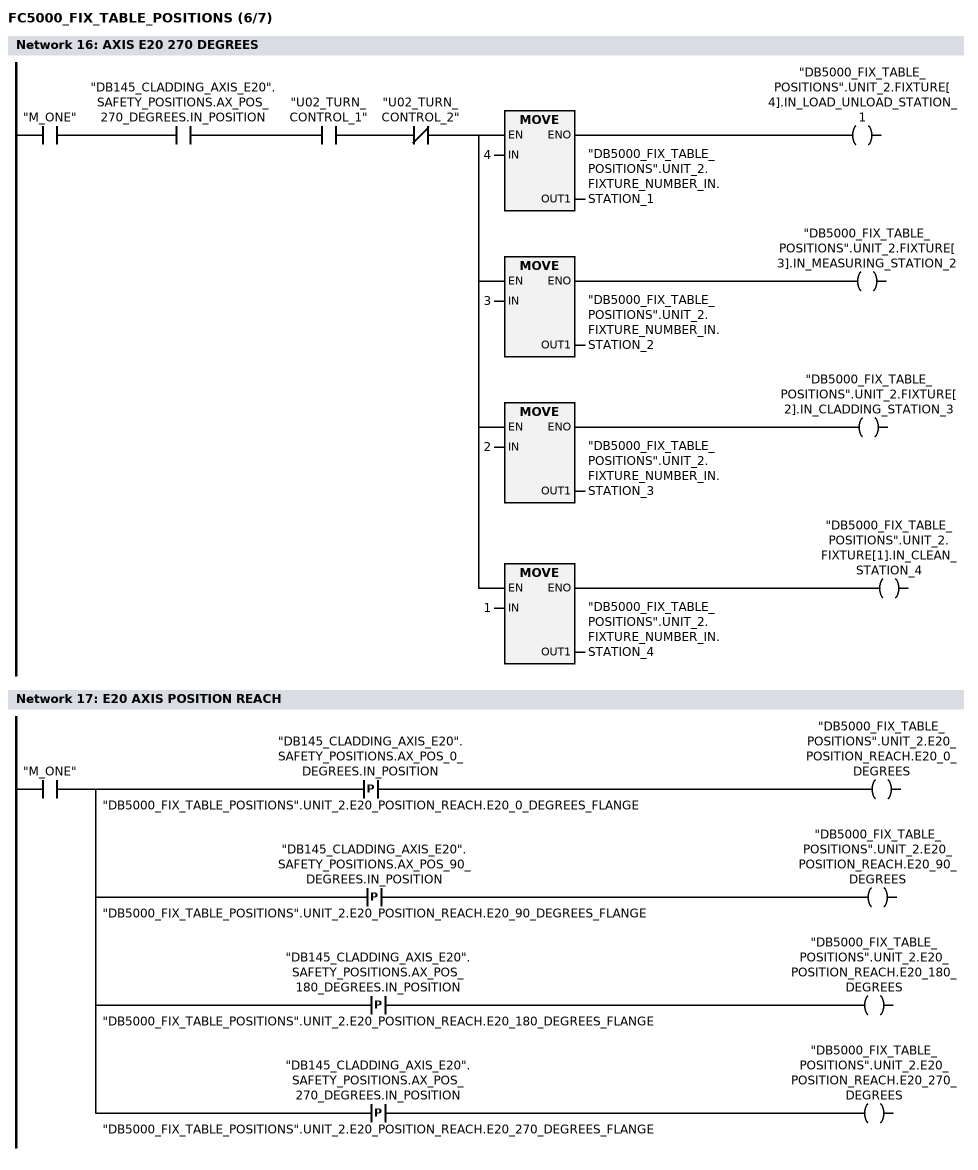
   RUNG wire#powerrail
      Contact( "M_ONE" )
      Contact( "DB145_CLADDING_AXIS_E20".SAFETY_POSITIONS.AX_POS_270_DEGREES.IN_POSITION )
      Contact( "U02_TURN_CONTROL_1" )
      I_Contact( "U02_TURN_CONTROL_2" )
      wire#w1
      Move(in := 4, out1 => "DB5000_FIX_TABLE_POSITIONS".UNIT_2.FIXTURE_NUMBER_IN.STATION_1)
      Coil( "DB5000_FIX_TABLE_POSITIONS".UNIT_2.FIXTURE[4].IN_LOAD_UNLOAD_STATION_1 )
   END_RUNG
   RUNG wire#w1
      Move(in := 3, out1 => "DB5000_FIX_TABLE_POSITIONS".UNIT_2.FIXTURE_NUMBER_IN.STATION_2)
      Coil( "DB5000_FIX_TABLE_POSITIONS".UNIT_2.FIXTURE[3].IN_MEASURING_STATION_2 )
   END_RUNG
   RUNG wire#w1
      Move(in := 2, out1 => "DB5000_FIX_TABLE_POSITIONS".UNIT_2.FIXTURE_NUMBER_IN.STATION_3)
      Coil( "DB5000_FIX_TABLE_POSITIONS".UNIT_2.FIXTURE[2].IN_CLADDING_STATION_3 )
   END_RUNG
   RUNG wire#w1
      Move(in := 1, out1 => "DB5000_FIX_TABLE_POSITIONS".UNIT_2.FIXTURE_NUMBER_IN.STATION_4)
      Coil( "DB5000_FIX_TABLE_POSITIONS".UNIT_2.FIXTURE[1].IN_CLEAN_STATION_4 )
   END_RUNG
   // the same network as SCL:
   #_w1 := "M_ONE" AND "DB145_CLADDING_AXIS_E20".SAFETY_POSITIONS.AX_POS_270_DEGREES.IN_POSITION AND "U02_TURN_CONTROL_1" AND NOT "U02_TURN_CONTROL_2";
   IF #_w1 THEN "DB5000_FIX_TABLE_POSITIONS".UNIT_2.FIXTURE_NUMBER_IN.STATION_1 := 4; END_IF;
   "DB5000_FIX_TABLE_POSITIONS".UNIT_2.FIXTURE[4].IN_LOAD_UNLOAD_STATION_1 := #_w1;
   IF #_w1 THEN "DB5000_FIX_TABLE_POSITIONS".UNIT_2.FIXTURE_NUMBER_IN.STATION_2 := 3; END_IF;
   "DB5000_FIX_TABLE_POSITIONS".UNIT_2.FIXTURE[3].IN_MEASURING_STATION_2 := #_w1;
   IF #_w1 THEN "DB5000_FIX_TABLE_POSITIONS".UNIT_2.FIXTURE_NUMBER_IN.STATION_3 := 2; END_IF;
   "DB5000_FIX_TABLE_POSITIONS".UNIT_2.FIXTURE[2].IN_CLADDING_STATION_3 := #_w1;
   IF #_w1 THEN "DB5000_FIX_TABLE_POSITIONS".UNIT_2.FIXTURE_NUMBER_IN.STATION_4 := 1; END_IF;
   "DB5000_FIX_TABLE_POSITIONS".UNIT_2.FIXTURE[1].IN_CLEAN_STATION_4 := #_w1;
END_REGION

REGION Network 17: E20 AXIS POSITION REACH
   RUNG wire#powerrail
      Contact( "M_ONE" )
      wire#w1
      P_Contact(operand := "DB145_CLADDING_AXIS_E20".SAFETY_POSITIONS.AX_POS_0_DEGREES.IN_POSITION, bit := "DB5000_FIX_TABLE_POSITIONS".UNIT_2.E20_POSITION_REACH.E20_0_DEGREES_FLANGE)
      Coil( "DB5000_FIX_TABLE_POSITIONS".UNIT_2.E20_POSITION_REACH.E20_0_DEGREES )
   END_RUNG
   RUNG wire#w1
      P_Contact(operand := "DB145_CLADDING_AXIS_E20".SAFETY_POSITIONS.AX_POS_90_DEGREES.IN_POSITION, bit := "DB5000_FIX_TABLE_POSITIONS".UNIT_2.E20_POSITION_REACH.E20_90_DEGREES_FLANGE)
      Coil( "DB5000_FIX_TABLE_POSITIONS".UNIT_2.E20_POSITION_REACH.E20_90_DEGREES )
   END_RUNG
   RUNG wire#w1
      P_Contact(operand := "DB145_CLADDING_AXIS_E20".SAFETY_POSITIONS.AX_POS_180_DEGREES.IN_POSITION, bit := "DB5000_FIX_TABLE_POSITIONS".UNIT_2.E20_POSITION_REACH.E20_180_DEGREES_FLANGE)
      Coil( "DB5000_FIX_TABLE_POSITIONS".UNIT_2.E20_POSITION_REACH.E20_180_DEGREES )
   END_RUNG
   RUNG wire#w1
      P_Contact(operand := "DB145_CLADDING_AXIS_E20".SAFETY_POSITIONS.AX_POS_270_DEGREES.IN_POSITION, bit := "DB5000_FIX_TABLE_POSITIONS".UNIT_2.E20_POSITION_REACH.E20_270_DEGREES_FLANGE)
      Coil( "DB5000_FIX_TABLE_POSITIONS".UNIT_2.E20_POSITION_REACH.E20_270_DEGREES )
   END_RUNG
   // the same network as SCL:
   #_w1 := "M_ONE" AND "DB145_CLADDING_AXIS_E20".SAFETY_POSITIONS.AX_POS_0_DEGREES.IN_POSITION AND NOT "DB5000_FIX_TABLE_POSITIONS".UNIT_2.E20_POSITION_REACH.E20_0_DEGREES_FLANGE;   // rising edge of "DB145_CLADDING_AXIS_E20".SAFETY_POSITIONS.AX_POS_0_DEGREES.IN_POSITION
   "DB5000_FIX_TABLE_POSITIONS".UNIT_2.E20_POSITION_REACH.E20_0_DEGREES_FLANGE := "DB145_CLADDING_AXIS_E20".SAFETY_POSITIONS.AX_POS_0_DEGREES.IN_POSITION;
   "DB5000_FIX_TABLE_POSITIONS".UNIT_2.E20_POSITION_REACH.E20_0_DEGREES := #_w1;
   #_w2 := "M_ONE" AND "DB145_CLADDING_AXIS_E20".SAFETY_POSITIONS.AX_POS_90_DEGREES.IN_POSITION AND NOT "DB5000_FIX_TABLE_POSITIONS".UNIT_2.E20_POSITION_REACH.E20_90_DEGREES_FLANGE;   // rising edge of "DB145_CLADDING_AXIS_E20".SAFETY_POSITIONS.AX_POS_90_DEGREES.IN_POSITION
   "DB5000_FIX_TABLE_POSITIONS".UNIT_2.E20_POSITION_REACH.E20_90_DEGREES_FLANGE := "DB145_CLADDING_AXIS_E20".SAFETY_POSITIONS.AX_POS_90_DEGREES.IN_POSITION;
   "DB5000_FIX_TABLE_POSITIONS".UNIT_2.E20_POSITION_REACH.E20_90_DEGREES := #_w2;
   #_w3 := "M_ONE" AND "DB145_CLADDING_AXIS_E20".SAFETY_POSITIONS.AX_POS_180_DEGREES.IN_POSITION AND NOT "DB5000_FIX_TABLE_POSITIONS".UNIT_2.E20_POSITION_REACH.E20_180_DEGREES_FLANGE;   // rising edge of "DB145_CLADDING_AXIS_E20".SAFETY_POSITIONS.AX_POS_180_DEGREES.IN_POSITION
   "DB5000_FIX_TABLE_POSITIONS".UNIT_2.E20_POSITION_REACH.E20_180_DEGREES_FLANGE := "DB145_CLADDING_AXIS_E20".SAFETY_POSITIONS.AX_POS_180_DEGREES.IN_POSITION;
   "DB5000_FIX_TABLE_POSITIONS".UNIT_2.E20_POSITION_REACH.E20_180_DEGREES := #_w3;
   #_w4 := "M_ONE" AND "DB145_CLADDING_AXIS_E20".SAFETY_POSITIONS.AX_POS_270_DEGREES.IN_POSITION AND NOT "DB5000_FIX_TABLE_POSITIONS".UNIT_2.E20_POSITION_REACH.E20_270_DEGREES_FLANGE;   // rising edge of "DB145_CLADDING_AXIS_E20".SAFETY_POSITIONS.AX_POS_270_DEGREES.IN_POSITION
   "DB5000_FIX_TABLE_POSITIONS".UNIT_2.E20_POSITION_REACH.E20_270_DEGREES_FLANGE := "DB145_CLADDING_AXIS_E20".SAFETY_POSITIONS.AX_POS_270_DEGREES.IN_POSITION;
   "DB5000_FIX_TABLE_POSITIONS".UNIT_2.E20_POSITION_REACH.E20_270_DEGREES := #_w4;
END_REGION

REGION Network 18: FIXTURES NO DEFINE POSITION
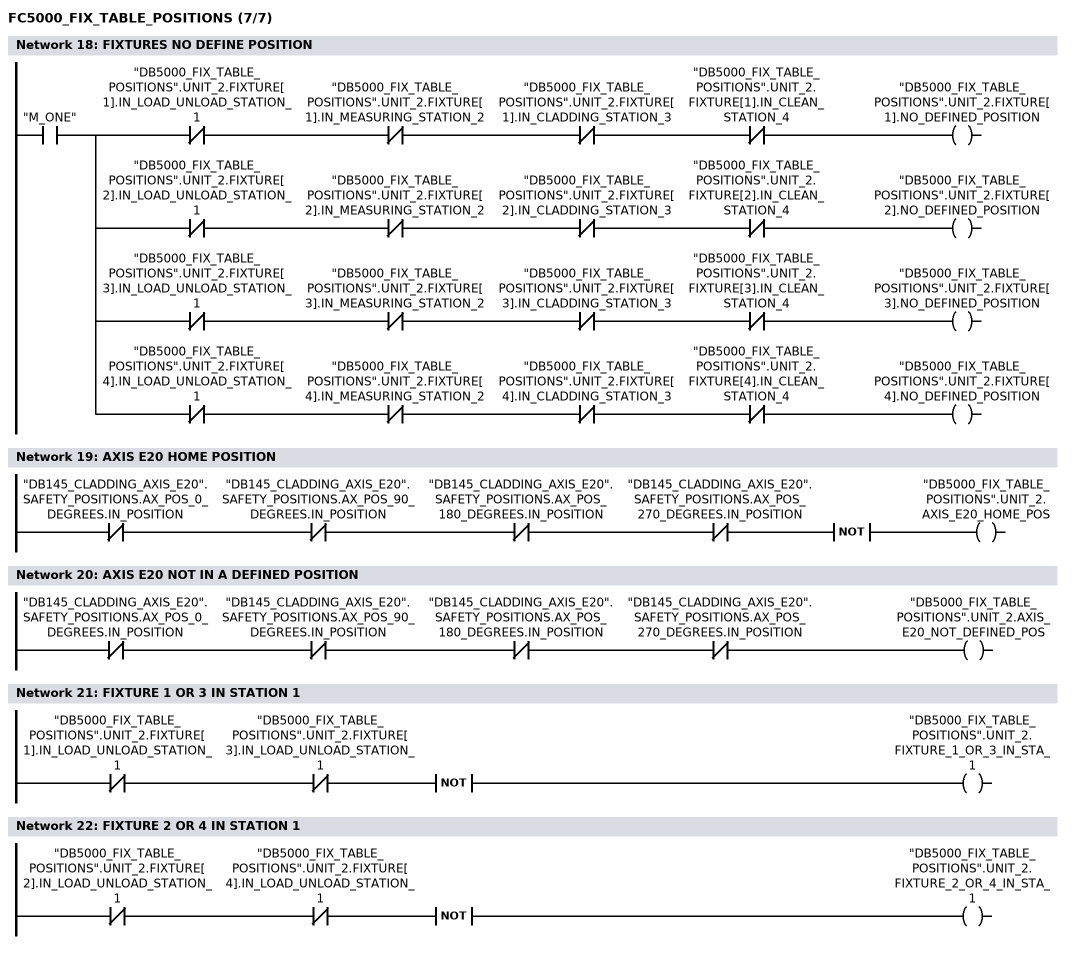
   RUNG wire#powerrail
      Contact( "M_ONE" )
      wire#w1
      I_Contact( "DB5000_FIX_TABLE_POSITIONS".UNIT_2.FIXTURE[1].IN_LOAD_UNLOAD_STATION_1 )
      I_Contact( "DB5000_FIX_TABLE_POSITIONS".UNIT_2.FIXTURE[1].IN_MEASURING_STATION_2 )
      I_Contact( "DB5000_FIX_TABLE_POSITIONS".UNIT_2.FIXTURE[1].IN_CLADDING_STATION_3 )
      I_Contact( "DB5000_FIX_TABLE_POSITIONS".UNIT_2.FIXTURE[1].IN_CLEAN_STATION_4 )
      Coil( "DB5000_FIX_TABLE_POSITIONS".UNIT_2.FIXTURE[1].NO_DEFINED_POSITION )
   END_RUNG
   RUNG wire#w1
      I_Contact( "DB5000_FIX_TABLE_POSITIONS".UNIT_2.FIXTURE[2].IN_LOAD_UNLOAD_STATION_1 )
      I_Contact( "DB5000_FIX_TABLE_POSITIONS".UNIT_2.FIXTURE[2].IN_MEASURING_STATION_2 )
      I_Contact( "DB5000_FIX_TABLE_POSITIONS".UNIT_2.FIXTURE[2].IN_CLADDING_STATION_3 )
      I_Contact( "DB5000_FIX_TABLE_POSITIONS".UNIT_2.FIXTURE[2].IN_CLEAN_STATION_4 )
      Coil( "DB5000_FIX_TABLE_POSITIONS".UNIT_2.FIXTURE[2].NO_DEFINED_POSITION )
   END_RUNG
   RUNG wire#w1
      I_Contact( "DB5000_FIX_TABLE_POSITIONS".UNIT_2.FIXTURE[3].IN_LOAD_UNLOAD_STATION_1 )
      I_Contact( "DB5000_FIX_TABLE_POSITIONS".UNIT_2.FIXTURE[3].IN_MEASURING_STATION_2 )
      I_Contact( "DB5000_FIX_TABLE_POSITIONS".UNIT_2.FIXTURE[3].IN_CLADDING_STATION_3 )
      I_Contact( "DB5000_FIX_TABLE_POSITIONS".UNIT_2.FIXTURE[3].IN_CLEAN_STATION_4 )
      Coil( "DB5000_FIX_TABLE_POSITIONS".UNIT_2.FIXTURE[3].NO_DEFINED_POSITION )
   END_RUNG
   RUNG wire#w1
      I_Contact( "DB5000_FIX_TABLE_POSITIONS".UNIT_2.FIXTURE[4].IN_LOAD_UNLOAD_STATION_1 )
      I_Contact( "DB5000_FIX_TABLE_POSITIONS".UNIT_2.FIXTURE[4].IN_MEASURING_STATION_2 )
      I_Contact( "DB5000_FIX_TABLE_POSITIONS".UNIT_2.FIXTURE[4].IN_CLADDING_STATION_3 )
      I_Contact( "DB5000_FIX_TABLE_POSITIONS".UNIT_2.FIXTURE[4].IN_CLEAN_STATION_4 )
      Coil( "DB5000_FIX_TABLE_POSITIONS".UNIT_2.FIXTURE[4].NO_DEFINED_POSITION )
   END_RUNG
   // the same network as SCL:
   "DB5000_FIX_TABLE_POSITIONS".UNIT_2.FIXTURE[1].NO_DEFINED_POSITION := "M_ONE" AND NOT "DB5000_FIX_TABLE_POSITIONS".UNIT_2.FIXTURE[1].IN_LOAD_UNLOAD_STATION_1 AND NOT "DB5000_FIX_TABLE_POSITIONS".UNIT_2.FIXTURE[1].IN_MEASURING_STATION_2 AND NOT "DB5000_FIX_TABLE_POSITIONS".UNIT_2.FIXTURE[1].IN_CLADDING_STATION_3 AND NOT "DB5000_FIX_TABLE_POSITIONS".UNIT_2.FIXTURE[1].IN_CLEAN_STATION_4;
   "DB5000_FIX_TABLE_POSITIONS".UNIT_2.FIXTURE[2].NO_DEFINED_POSITION := "M_ONE" AND NOT "DB5000_FIX_TABLE_POSITIONS".UNIT_2.FIXTURE[2].IN_LOAD_UNLOAD_STATION_1 AND NOT "DB5000_FIX_TABLE_POSITIONS".UNIT_2.FIXTURE[2].IN_MEASURING_STATION_2 AND NOT "DB5000_FIX_TABLE_POSITIONS".UNIT_2.FIXTURE[2].IN_CLADDING_STATION_3 AND NOT "DB5000_FIX_TABLE_POSITIONS".UNIT_2.FIXTURE[2].IN_CLEAN_STATION_4;
   "DB5000_FIX_TABLE_POSITIONS".UNIT_2.FIXTURE[3].NO_DEFINED_POSITION := "M_ONE" AND NOT "DB5000_FIX_TABLE_POSITIONS".UNIT_2.FIXTURE[3].IN_LOAD_UNLOAD_STATION_1 AND NOT "DB5000_FIX_TABLE_POSITIONS".UNIT_2.FIXTURE[3].IN_MEASURING_STATION_2 AND NOT "DB5000_FIX_TABLE_POSITIONS".UNIT_2.FIXTURE[3].IN_CLADDING_STATION_3 AND NOT "DB5000_FIX_TABLE_POSITIONS".UNIT_2.FIXTURE[3].IN_CLEAN_STATION_4;
   "DB5000_FIX_TABLE_POSITIONS".UNIT_2.FIXTURE[4].NO_DEFINED_POSITION := "M_ONE" AND NOT "DB5000_FIX_TABLE_POSITIONS".UNIT_2.FIXTURE[4].IN_LOAD_UNLOAD_STATION_1 AND NOT "DB5000_FIX_TABLE_POSITIONS".UNIT_2.FIXTURE[4].IN_MEASURING_STATION_2 AND NOT "DB5000_FIX_TABLE_POSITIONS".UNIT_2.FIXTURE[4].IN_CLADDING_STATION_3 AND NOT "DB5000_FIX_TABLE_POSITIONS".UNIT_2.FIXTURE[4].IN_CLEAN_STATION_4;
END_REGION

REGION Network 19: AXIS E20 HOME POSITION
   RUNG wire#powerrail
      I_Contact( "DB145_CLADDING_AXIS_E20".SAFETY_POSITIONS.AX_POS_0_DEGREES.IN_POSITION )
      I_Contact( "DB145_CLADDING_AXIS_E20".SAFETY_POSITIONS.AX_POS_90_DEGREES.IN_POSITION )
      I_Contact( "DB145_CLADDING_AXIS_E20".SAFETY_POSITIONS.AX_POS_180_DEGREES.IN_POSITION )
      I_Contact( "DB145_CLADDING_AXIS_E20".SAFETY_POSITIONS.AX_POS_270_DEGREES.IN_POSITION )
      Not()
      Coil( "DB5000_FIX_TABLE_POSITIONS".UNIT_2.AXIS_E20_HOME_POS )
   END_RUNG
   // the same network as SCL:
   "DB5000_FIX_TABLE_POSITIONS".UNIT_2.AXIS_E20_HOME_POS := NOT (NOT "DB145_CLADDING_AXIS_E20".SAFETY_POSITIONS.AX_POS_0_DEGREES.IN_POSITION AND NOT "DB145_CLADDING_AXIS_E20".SAFETY_POSITIONS.AX_POS_90_DEGREES.IN_POSITION AND NOT "DB145_CLADDING_AXIS_E20".SAFETY_POSITIONS.AX_POS_180_DEGREES.IN_POSITION AND NOT "DB145_CLADDING_AXIS_E20".SAFETY_POSITIONS.AX_POS_270_DEGREES.IN_POSITION);
END_REGION

REGION Network 20: AXIS E20 NOT IN A DEFINED POSITION
   RUNG wire#powerrail
      I_Contact( "DB145_CLADDING_AXIS_E20".SAFETY_POSITIONS.AX_POS_0_DEGREES.IN_POSITION )
      I_Contact( "DB145_CLADDING_AXIS_E20".SAFETY_POSITIONS.AX_POS_90_DEGREES.IN_POSITION )
      I_Contact( "DB145_CLADDING_AXIS_E20".SAFETY_POSITIONS.AX_POS_180_DEGREES.IN_POSITION )
      I_Contact( "DB145_CLADDING_AXIS_E20".SAFETY_POSITIONS.AX_POS_270_DEGREES.IN_POSITION )
      Coil( "DB5000_FIX_TABLE_POSITIONS".UNIT_2.AXIS_E20_NOT_DEFINED_POS )
   END_RUNG
   // the same network as SCL:
   "DB5000_FIX_TABLE_POSITIONS".UNIT_2.AXIS_E20_NOT_DEFINED_POS := NOT "DB145_CLADDING_AXIS_E20".SAFETY_POSITIONS.AX_POS_0_DEGREES.IN_POSITION AND NOT "DB145_CLADDING_AXIS_E20".SAFETY_POSITIONS.AX_POS_90_DEGREES.IN_POSITION AND NOT "DB145_CLADDING_AXIS_E20".SAFETY_POSITIONS.AX_POS_180_DEGREES.IN_POSITION AND NOT "DB145_CLADDING_AXIS_E20".SAFETY_POSITIONS.AX_POS_270_DEGREES.IN_POSITION;
END_REGION

REGION Network 21: FIXTURE 1 OR 3 IN STATION 1
   RUNG wire#powerrail
      I_Contact( "DB5000_FIX_TABLE_POSITIONS".UNIT_2.FIXTURE[1].IN_LOAD_UNLOAD_STATION_1 )
      I_Contact( "DB5000_FIX_TABLE_POSITIONS".UNIT_2.FIXTURE[3].IN_LOAD_UNLOAD_STATION_1 )
      Not()
      Coil( "DB5000_FIX_TABLE_POSITIONS".UNIT_2.FIXTURE_1_OR_3_IN_STA_1 )
   END_RUNG
   // the same network as SCL:
   "DB5000_FIX_TABLE_POSITIONS".UNIT_2.FIXTURE_1_OR_3_IN_STA_1 := NOT (NOT "DB5000_FIX_TABLE_POSITIONS".UNIT_2.FIXTURE[1].IN_LOAD_UNLOAD_STATION_1 AND NOT "DB5000_FIX_TABLE_POSITIONS".UNIT_2.FIXTURE[3].IN_LOAD_UNLOAD_STATION_1);
END_REGION

REGION Network 22: FIXTURE 2 OR 4 IN STATION 1
   RUNG wire#powerrail
      I_Contact( "DB5000_FIX_TABLE_POSITIONS".UNIT_2.FIXTURE[2].IN_LOAD_UNLOAD_STATION_1 )
      I_Contact( "DB5000_FIX_TABLE_POSITIONS".UNIT_2.FIXTURE[4].IN_LOAD_UNLOAD_STATION_1 )
      Not()
      Coil( "DB5000_FIX_TABLE_POSITIONS".UNIT_2.FIXTURE_2_OR_4_IN_STA_1 )
   END_RUNG
   // the same network as SCL:
   "DB5000_FIX_TABLE_POSITIONS".UNIT_2.FIXTURE_2_OR_4_IN_STA_1 := NOT (NOT "DB5000_FIX_TABLE_POSITIONS".UNIT_2.FIXTURE[2].IN_LOAD_UNLOAD_STATION_1 AND NOT "DB5000_FIX_TABLE_POSITIONS".UNIT_2.FIXTURE[4].IN_LOAD_UNLOAD_STATION_1);
END_REGION
END_FUNCTION
